TYPE E_DCH_Error :
(
	None,
	Unknown,
	MAX_E_DCH_Error
);
END_TYPE

(* stored: Version 1.1.0.1, ProductVersion 3.1.0.26
   DUT E_DCH_Error: Id {d1441eaa-43a8-4439-b7ea-f1711ceb1e2b} *)
